SUBAPPLICATION AuxPic (* Bild- und Farbumschaltung für AUX-N und VT Objekte *)
  (* Standard: 61499-2 *)
  (* Version 1.1, 2026-04-09, Christoph Behr, HR Agrartechnik, Inits verbunden und REQ angeschlossen *)
  (* Version 1.0, 2025-06-12, franz *)
  PACKAGE MyLib::sys;
  IMPORT logiBUS::utils::sequence::schieber::SchieberAuxOutStruct;
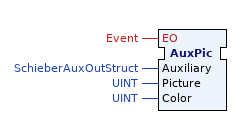
  EVENT_INPUT
    EO;
  END_EVENT
  VAR_INPUT
    Auxiliary : logiBUS::utils::sequence::schieber::SchieberAuxOutStruct;
    Picture : UINT; (* Object ID of the ObjectPointer to the Picture *)
    Color : UINT; (* Object ID of the AuxFunction *)
  END_VAR
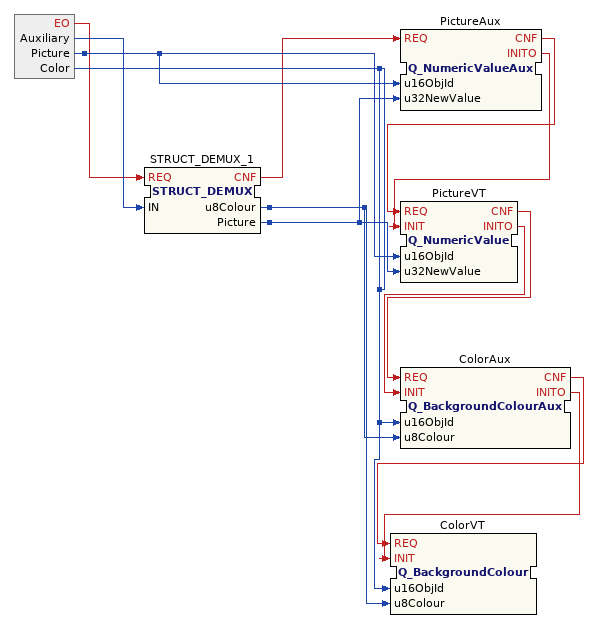
  FBS
    PictureVT : isobus::UT::Q::Q_NumericValue;
    ColorAux : isobus::UT::Q::Q_BackgroundColourAux;
    PictureAux : isobus::UT::Q::Q_NumericValueAux;
    ColorVT : isobus::UT::Q::Q_BackgroundColour;
    STRUCT_DEMUX_1 : eclipse4diac::convert::STRUCT_DEMUX; {SET_ATTRIBUTE(StructuredType, logiBUS::utils::sequence::schieber::SchieberAuxOutStruct)}
  END_FBS
  EVENT_CONNECTIONS
    EO TO STRUCT_DEMUX_1.REQ;
    STRUCT_DEMUX_1.CNF TO PictureAux.REQ;
    PictureAux.CNF TO PictureVT.REQ;
    PictureVT.CNF TO ColorAux.REQ;
    ColorAux.CNF TO ColorVT.REQ;
    PictureAux.INITO TO PictureVT.INIT;
    PictureVT.INITO TO ColorAux.INIT;
    ColorAux.INITO TO ColorVT.INIT;
  END_CONNECTIONS
  DATA_CONNECTIONS
    Color TO ColorAux.u16ObjId;
    Color TO ColorVT.u16ObjId;
    Picture TO PictureAux.u16ObjId;
    Picture TO PictureVT.u16ObjId;
    Auxiliary TO STRUCT_DEMUX_1.IN;
    STRUCT_DEMUX_1.u8Colour TO ColorVT.u8Colour;
    STRUCT_DEMUX_1.u8Colour TO ColorAux.u8Colour;
    STRUCT_DEMUX_1.Picture TO PictureAux.u32NewValue;
    STRUCT_DEMUX_1.Picture TO PictureVT.u32NewValue;
  END_CONNECTIONS
END_SUBAPPLICATION
